// Mitsubishi GX Works2 project: MOVE비트관리   PLC: Q02/Q02H

PROGRAM MAIN
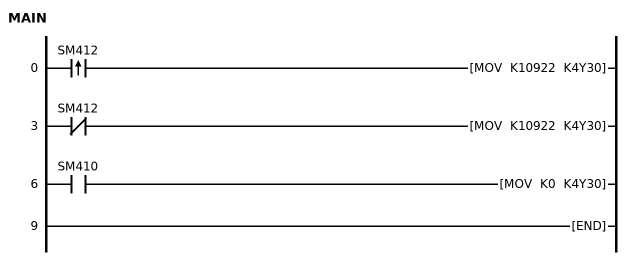
0     LDP     SM412
      MOV     K10922 K4Y30
3     LDI     SM412
      MOV     K10922 K4Y30
6     LD      SM410
      MOV     K0 K4Y30
9     END
END_PROGRAM
